{attribute addProperty BoxType "EK1122-0000-0018"}
{attribute addProperty Id "Beckhoff_EP7xxxsub_EK1100EK1100_179A0949162A_0001_EP7041_0002_0016EP7041_48B7DF6040750.875A_0002_EP7041_0002_0017EP7041_48B7DF6040750.875A_0003_EP7041_0002_0018EP7041_8145D2A024030A_0004_EP7041_0002_0019EP7041_8145D2A024030A_0005_EP7041_0002_0020EP7041_8145D2A024030A_0006_EP7041_0002_0021EP7041_8145D2A024030A_0007_EP7041_0002_0022EP7041_8145D2A024030A_0008_EP7041_0002_0023EP7041_5614098424030A_0009_EP7041_0002_0024EP7041_5614098424030A_0010_EP7041_0002_0025EP7041_5614098424030A_0011_EP7041_1002_0017EP7041_48B7DF6040750.875A_0012_EP7041_1002_0018EP7041_8145D2A024030A_0013_EP7041_1002_0019EP7041_8145D2A024030A_0014_EP7041_1002_0020EP7041_8145D2A024030A_0015_EP7041_1002_0021EP7041_8145D2A024030A_0016_EP7041_1002_0022EP7041_8145D2A024030A_0017_EP7041_1002_0023EP7041_5614098424030A_0018_EP7041_1002_0024EP7041_5614098424030A_0019_EP7041_1002_0025EP7041_5614098424030A_0020_EP7041_2002_0016EP7041_8145D2A024030A_0021_EP7041_2002_0019EP7041_8145D2A024030A_0022_EP7041_2002_0020EP7041_8145D2A024030A_0023_EP7041_2002_0021EP7041_8145D2A024030A_0024_EP7041_2002_0022EP7041_8145D2A024030A_0025_EP7041_2002_0023EP7041_5614098424030A_0026_EP7041_2002_0024EP7041_5614098424030A_0027_EP7041_2002_0025EP7041_5614098424030A_0028_EP7041_3002_0016EP7041_8ADDF8F224030A_0029_EP7041_3002_0017EP7041_8ADDF8F224030A_0030_EP7041_3002_0018EP7041_8ADDF8F224030A_0031_EP7041_3002_0019EP7041_8ADDF8F224030A_0032_EP7041_3002_0020EP7041_E93814AC24030A_0033_EP7041_3002_0021EP7041_E93814AC24030A_0034_EP7041_3002_0022EP7041_E93814AC24030A_0035_EP7041_3102_0016EP7041_E93814AC24030A_0036_EP7041_3102_0017EP7041_E93814AC24030A_0037_EP7041_3102_0022EP7041_E93814AC24030A_0038_EP7047_1032_0021EP7047_E93814AC24030A_0039_EP7211_0034_0029EP7211_5C47483126433A_0040_EP7211_0034_0030EP7211_F2E8196327234A_0041_EP7211_0034_0031EP7211_F2E8196327234A_0042_EP7211_0034_0032EP7211_F2E8196327234A_0043_EP7211_0035_0029EP7211_A058FB7326433A_0044_EP7211_0035_0030EP7211_A058FB7326433A_0045_EP7211_0035_0031EP7211_A058FB7326433A_0046_EP7211_0035_0032EP7211_A058FB7326433A_0047_EP7342_0002_0016EP7342_5DC6D75238448A_0048_EP7342_0002_0017EP7342_5DC6D75238448A_0049_EP7342_0002_0018EP7342_5DC6D75238448A_0050_EP7342_0002_0019EP7342_5DC6D75238448A_0051_EP7342_0002_0020EP7342_5DC6D75238448A_0052_EP7342_0002_0021EP7342_014E044838448A_0053_EP7342_0002_0022EP7342_014E044838448A_0054_EP7402_0057_0017A_0054_EP7402_0057_0017_44AF23AC54468"}
{attribute addProperty CRC "3454385400"}
{attribute addProperty SizeInBites "15005"}
{attribute addProperty SizeInBytes "1875.625"}
TYPE Beckhoff_EP7xxxEK1122_CDE5BCF8 EXTENDS EK1122_179A0949 :
STRUCT
	{attribute addProperty Name "Beckhoff_EP7xxxsub_EK1100"}
	Beckhoff_EP7xxxsub_EK1100 : EK1100_179A0949;
	{attribute addProperty Name "A_0001_EP7041_0002_0016"}
	A_0001_EP7041_0002_0016 : EP7041_48B7DF60;
	{attribute addProperty Name "A_0002_EP7041_0002_0017"}
	A_0002_EP7041_0002_0017 : EP7041_48B7DF60;
	{attribute addProperty Name "A_0003_EP7041_0002_0018"}
	A_0003_EP7041_0002_0018 : EP7041_8145D2A0;
	{attribute addProperty Name "A_0004_EP7041_0002_0019"}
	A_0004_EP7041_0002_0019 : EP7041_8145D2A0;
	{attribute addProperty Name "A_0005_EP7041_0002_0020"}
	A_0005_EP7041_0002_0020 : EP7041_8145D2A0;
	{attribute addProperty Name "A_0006_EP7041_0002_0021"}
	A_0006_EP7041_0002_0021 : EP7041_8145D2A0;
	{attribute addProperty Name "A_0007_EP7041_0002_0022"}
	A_0007_EP7041_0002_0022 : EP7041_8145D2A0;
	{attribute addProperty Name "A_0008_EP7041_0002_0023"}
	A_0008_EP7041_0002_0023 : EP7041_56140984;
	{attribute addProperty Name "A_0009_EP7041_0002_0024"}
	A_0009_EP7041_0002_0024 : EP7041_56140984;
	{attribute addProperty Name "A_0010_EP7041_0002_0025"}
	A_0010_EP7041_0002_0025 : EP7041_56140984;
	{attribute addProperty Name "A_0011_EP7041_1002_0017"}
	A_0011_EP7041_1002_0017 : EP7041_48B7DF60;
	{attribute addProperty Name "A_0012_EP7041_1002_0018"}
	A_0012_EP7041_1002_0018 : EP7041_8145D2A0;
	{attribute addProperty Name "A_0013_EP7041_1002_0019"}
	A_0013_EP7041_1002_0019 : EP7041_8145D2A0;
	{attribute addProperty Name "A_0014_EP7041_1002_0020"}
	A_0014_EP7041_1002_0020 : EP7041_8145D2A0;
	{attribute addProperty Name "A_0015_EP7041_1002_0021"}
	A_0015_EP7041_1002_0021 : EP7041_8145D2A0;
	{attribute addProperty Name "A_0016_EP7041_1002_0022"}
	A_0016_EP7041_1002_0022 : EP7041_8145D2A0;
	{attribute addProperty Name "A_0017_EP7041_1002_0023"}
	A_0017_EP7041_1002_0023 : EP7041_56140984;
	{attribute addProperty Name "A_0018_EP7041_1002_0024"}
	A_0018_EP7041_1002_0024 : EP7041_56140984;
	{attribute addProperty Name "A_0019_EP7041_1002_0025"}
	A_0019_EP7041_1002_0025 : EP7041_56140984;
	{attribute addProperty Name "A_0020_EP7041_2002_0016"}
	A_0020_EP7041_2002_0016 : EP7041_8145D2A0;
	{attribute addProperty Name "A_0021_EP7041_2002_0019"}
	A_0021_EP7041_2002_0019 : EP7041_8145D2A0;
	{attribute addProperty Name "A_0022_EP7041_2002_0020"}
	A_0022_EP7041_2002_0020 : EP7041_8145D2A0;
	{attribute addProperty Name "A_0023_EP7041_2002_0021"}
	A_0023_EP7041_2002_0021 : EP7041_8145D2A0;
	{attribute addProperty Name "A_0024_EP7041_2002_0022"}
	A_0024_EP7041_2002_0022 : EP7041_8145D2A0;
	{attribute addProperty Name "A_0025_EP7041_2002_0023"}
	A_0025_EP7041_2002_0023 : EP7041_56140984;
	{attribute addProperty Name "A_0026_EP7041_2002_0024"}
	A_0026_EP7041_2002_0024 : EP7041_56140984;
	{attribute addProperty Name "A_0027_EP7041_2002_0025"}
	A_0027_EP7041_2002_0025 : EP7041_56140984;
	{attribute addProperty Name "A_0028_EP7041_3002_0016"}
	A_0028_EP7041_3002_0016 : EP7041_8ADDF8F2;
	{attribute addProperty Name "A_0029_EP7041_3002_0017"}
	A_0029_EP7041_3002_0017 : EP7041_8ADDF8F2;
	{attribute addProperty Name "A_0030_EP7041_3002_0018"}
	A_0030_EP7041_3002_0018 : EP7041_8ADDF8F2;
	{attribute addProperty Name "A_0031_EP7041_3002_0019"}
	A_0031_EP7041_3002_0019 : EP7041_8ADDF8F2;
	{attribute addProperty Name "A_0032_EP7041_3002_0020"}
	A_0032_EP7041_3002_0020 : EP7041_E93814AC;
	{attribute addProperty Name "A_0033_EP7041_3002_0021"}
	A_0033_EP7041_3002_0021 : EP7041_E93814AC;
	{attribute addProperty Name "A_0034_EP7041_3002_0022"}
	A_0034_EP7041_3002_0022 : EP7041_E93814AC;
	{attribute addProperty Name "A_0035_EP7041_3102_0016"}
	A_0035_EP7041_3102_0016 : EP7041_E93814AC;
	{attribute addProperty Name "A_0036_EP7041_3102_0017"}
	A_0036_EP7041_3102_0017 : EP7041_E93814AC;
	{attribute addProperty Name "A_0037_EP7041_3102_0022"}
	A_0037_EP7041_3102_0022 : EP7041_E93814AC;
	{attribute addProperty Name "A_0038_EP7047_1032_0021"}
	A_0038_EP7047_1032_0021 : EP7047_E93814AC;
	{attribute addProperty Name "A_0039_EP7211_0034_0029"}
	A_0039_EP7211_0034_0029 : EP7211_5C474831;
	{attribute addProperty Name "A_0040_EP7211_0034_0030"}
	A_0040_EP7211_0034_0030 : EP7211_F2E81963;
	{attribute addProperty Name "A_0041_EP7211_0034_0031"}
	A_0041_EP7211_0034_0031 : EP7211_F2E81963;
	{attribute addProperty Name "A_0042_EP7211_0034_0032"}
	A_0042_EP7211_0034_0032 : EP7211_F2E81963;
	{attribute addProperty Name "A_0043_EP7211_0035_0029"}
	A_0043_EP7211_0035_0029 : EP7211_A058FB73;
	{attribute addProperty Name "A_0044_EP7211_0035_0030"}
	A_0044_EP7211_0035_0030 : EP7211_A058FB73;
	{attribute addProperty Name "A_0045_EP7211_0035_0031"}
	A_0045_EP7211_0035_0031 : EP7211_A058FB73;
	{attribute addProperty Name "A_0046_EP7211_0035_0032"}
	A_0046_EP7211_0035_0032 : EP7211_A058FB73;
	{attribute addProperty Name "A_0047_EP7342_0002_0016"}
	A_0047_EP7342_0002_0016 : EP7342_5DC6D752;
	{attribute addProperty Name "A_0048_EP7342_0002_0017"}
	A_0048_EP7342_0002_0017 : EP7342_5DC6D752;
	{attribute addProperty Name "A_0049_EP7342_0002_0018"}
	A_0049_EP7342_0002_0018 : EP7342_5DC6D752;
	{attribute addProperty Name "A_0050_EP7342_0002_0019"}
	A_0050_EP7342_0002_0019 : EP7342_5DC6D752;
	{attribute addProperty Name "A_0051_EP7342_0002_0020"}
	A_0051_EP7342_0002_0020 : EP7342_5DC6D752;
	{attribute addProperty Name "A_0052_EP7342_0002_0021"}
	A_0052_EP7342_0002_0021 : EP7342_014E0448;
	{attribute addProperty Name "A_0053_EP7342_0002_0022"}
	A_0053_EP7342_0002_0022 : EP7342_014E0448;
	{attribute addProperty Name "A_0054_EP7402_0057_0017"}
	A_0054_EP7402_0057_0017 : A_0054_EP7402_0057_0017_44AF23AC;
END_STRUCT
END_TYPE

(* stored: Version 1.2.0.0, ProductVersion 3.1.4024.9
   DUT Beckhoff_EP7xxxEK1122_CDE5BCF8: Id {65d2cf5a-9ae8-4d0f-87df-19514404adb4} *)
